// TwinCAT 3 PLC project Untitled1
// ProgramVersion: 3.1.4023.0
// libraries:
//   Tc2_Standard, * (Beckhoff Automation GmbH)
//   Tc2_System, * (Beckhoff Automation GmbH)
//   Tc2_Utilities, * (Beckhoff Automation GmbH)
//   Tc3_IotBase, * (Beckhoff Automation GmbH)
//   Tc3_Module, * (Beckhoff Automation GmbH)
// project tree:
//   DUTs/ MQTTSettings.TcDUT
//   / PlcTask.TcTTO (not stored)
//   POUs/ MAIN.TcPOU, MQTT.TcPOU
// real-time tasks:
//   TASK PlcTask: cycle T#10ms, priority 20, ADS port 350

// ---- DUTs/MQTTSettings.TcDUT
TYPE MQTTSettings :
STRUCT
	//Broker info
	brokerIP : STRING := '78.27.125.143';
    brokerPort : UINT := 8885;
	brokerUsername : STRING := 'scanrobot';
	brokerPassword : STRING := 'kissa';
	
	//Client info
    clientId : STRING := 'plc';
	topicPub : STRING := 'beckhoff';
	topicSub : STRING := 'plc';
	qos : TcIotMqttQos := TcIotMqttQos.AtMostOnceDelivery;	
	
	//TLS info
	caCertificateAbsolutePath : STRING := 'C:\Users\mikko\Desktop\twincat\certs\ca.crt';
	clientCertificateAbsolutePath : STRING := 'C:\Users\mikko\Desktop\twincat\certs\client.crt';
	clientKeyAbsolutePath : STRING := 'C:\Users\mikko\Desktop\twincat\certs\client.key';
END_STRUCT
END_TYPE

// ---- POUs/MAIN.TcPOU
PROGRAM MAIN
VAR
	mqtt: MQTT;
	
	tonTimer : TON := (PT:=T#1S); //Interval timer for broadcasting.
	counter : INT := 0;
	isPublished : BOOL := FALSE;
END_VAR

IF _TaskInfo[GETCURTASKINDEXEX()].FirstCycle THEN
	mqtt.configureMQTTClient();
END_IF 
mqtt.connect();

IF mqtt.isConnected() THEN
	//Capasity test
	IF NOT isPublished THEN
		mqtt.publish(msg := 'this is a very long message for testing mqtt maximum capacity. this is a very lo');
		isPublished := TRUE;
	END_IF

	
	
    //tonTimer(IN:=TRUE);
    //IF tonTimer.Q THEN
		//msg test
		//mqtt.publish(msg := '{"temperature":345;"motorSpeed":300;"distance":1345;"humidity":58}');
	
	
		//counter test
		//counter := counter + 1;		
        //tonTimer(IN:=FALSE);  
        //mqtt.publish(msg := TO_STRING(counter));
    //END_IF
	
END_IF

END_PROGRAM

// ---- POUs/MQTT.TcPOU
FUNCTION_BLOCK MQTT
VAR_OUTPUT
	mqttClient : FB_IotMqttClient;
END_VAR
VAR
	mqttSettings : MQTTSettings;
	messageQueue : FB_IotMqttMessageQueue;
    message      : FB_IotMqttMessage;
	isSubscribed : BOOL;
END_VAR

METHOD PUBLIC configureMQTTClient
VAR_IN_OUT
END_VAR
mqttClient.sHostName := mqttSettings.brokerIP;
mqttClient.nHostPort := mqttSettings.brokerPort;
mqttClient.sClientId := mqttSettings.clientId;
mqttClient.sUserName := mqttSettings.brokerUsername;
mqttClient.sUserPassword := mqttSettings.brokerPassword;
mqttClient.stTLS.sCA := mqttSettings.caCertificateAbsolutePath;
mqttClient.stTLS.sCert := mqttSettings.clientCertificateAbsolutePath;
mqttClient.stTLS.sKeyFile := mqttSettings.clientKeyAbsolutePath;
END_METHOD

METHOD PUBLIC connect
mqttClient.Execute(bConnect := TRUE);
END_METHOD

METHOD PUBLIC isConnected : BOOL
isConnected := mqttClient.bConnected;
END_METHOD

METHOD PUBLIC publish : BOOL
VAR_INPUT
	msg : STRING;
END_VAR
mqttClient.Publish(sTopic:= mqttSettings.topicPub,
            pPayload:= ADR(msg),
            nPayloadSize:= LEN2(ADR(msg))+1,
            eQoS:= mqttSettings.qos,
            bRetain:= FALSE,
            bQueue:= FALSE
);
END_METHOD

METHOD publishBack : BOOL
VAR_INPUT
END_VAR
VAR
	receivedTopic : STRING(255);
	receivedMsg : STRING(255);
END_VAR
IF isConnected() THEN
	IF NOT isSubscribed THEN
        isSubscribed := mqttClient.Subscribe(sTopic:=mqttSettings.topicSub, eQoS:=mqttSettings.qos);
		publish(msg := 'now subscribed!');
		publish(msg := mqttSettings.topicSub);
    END_IF	

	IF messageQueue.nQueuedMessages > 0 THEN
		publish(msg := 'something received');
		
		IF messageQueue.Dequeue(fbMessage:=message) THEN
			message.GetTopic(pTopic:=ADR(receivedTopic), nTopicSize:=SIZEOF(receivedTopic) );
			message.GetPayload(pPayload:=ADR(receivedMsg), nPayloadSize:=SIZEOF(receivedMsg), bSetNullTermination:=FALSE);
						
			publish(msg := receivedTopic);
			publish(msg := receivedMsg);
		END_IF
	END_IF
	
END_IF
END_METHOD

METHOD PUBLIC publishWithTON
VAR_IN_OUT
	timer : TON;	
END_VAR
VAR_INPUT
	msg : STRING;
END_VAR
IF isConnected() THEN
    timer(IN:=TRUE);
    IF timer.Q THEN
        timer(IN:=FALSE);
     
        publish(msg := msg);
    END_IF
END_IF
END_METHOD

END_FUNCTION_BLOCK
